PROGRAM P11_E3508
VAR_INPUT
	nTemperatureTargetValue	: INT(0..1200); //Target Values, Input Range 0 ~ 1200 Celcius
	nRampTime				: INT := 1; //Second
	nPowerRateSetValue		: WORD;	
	bOutputManAuto 			: BOOL; // 0:Auto, 1:Manual Operation
	
	bHeaterOn				: BOOL := FALSE; //to PSTEK
	bHeaterReset			: BOOL; //to PSTEK

END_VAR
VAR_OUTPUT
	bAlarmState_E3508 		: BOOL; //Alarm or Sensor Break Signal
	bManAuto_E3508 			: BOOL; // 0:Manual, 1:Auto
	rPowerRate				: REAL;	//Power rate for Monitoring
	
	isHeaterReady			: BOOL; //Close : Ready
	isHeaterRun				: BOOL; //Close : Running, Open : Stop
	isHeaterFault			: BOOL; //Close : Falut, Open : Normal
	//isInductionHeaterErr	: BOOL; //Power Supply
	bInductionHeaterCB		: BOOL;
END_VAR

VAR
	//Input from E3508 Controller
	aInputPVBytes AT %I* 		: ARRAY[1..2]OF USINT; //Input Process Values
	aInputSVBytes AT %I* 		: ARRAY[1..2]OF USINT; //Input Set Values
	aInputTVBytes AT %I* 		: ARRAY[1..2]OF USINT; //Input Target Valuse
	aInputCVBytes AT %I* 		: ARRAY[1..2]OF USINT; //Induction Heter Controlled Values
	aInputProportional AT %I* 	: ARRAY[1..2]OF USINT; //PID - Proportional Band
	aInputIntegral AT %I* 		: ARRAY[1..2]OF USINT; //PID - Integral Time
	aInputDerivative AT %I* 	: ARRAY[1..2]OF USINT; //PID - Derivative Time 
	nInputAlarmBytes AT %I* 	: USINT; // Alarm State
	nInputManAutoBytes AT %I* 	: USINT; // ManAuto State
	
	nTemperaturePV_E3508		: WORD;
	nTemperatureSV_E3508		: WORD;
	nPowerRate_E3508		: WORD; //To Induction Heater Control Values
	nParameterP				: WORD; //PID Parameter P
	nParameterI				: WORD; //PID Parameter I
	nParameterD				: WORD; //PID Parameter D
	//Output to E3508 Controller
	wOutputSVBytes 				: outWord;
	wOutputPowerSVBytes 		: outWord;
	aOutputSVBytes AT %Q* 		: ARRAY[1..2]OF USINT; //Temperature Set Value
	nOutputManAutoBytes AT %Q* 	: USINT; //ManAuto Change
	aOutputPowerBytes AT %Q* 	: ARRAY[1..2]OF USINT; //Output Power in Manual State
	//nOutputAlarmClear AT %Q* : USINT; //Alarm Clear Set
	
	nTemperatureControlValue	: WORD;
	
	// for FB_CTRL_RAMP_GENERATOR Variable
	(* input *)
	bEnable					: BOOL;
	rTemperatureStartValue	: REAL;
	rTemperatureTargetValue	: REAL;
	(* output *)
	rTemperatureControlValue : LREAL;
	bValueReached			: BOOL;
	(* function block *)
	fbCTRL_RAMP_GENERATOR		: FB_CTRL_RAMP_GENERATOR;
	stCTRL_RAMP_GENERATOR_PARAMS: ST_CTRL_RAMP_GENERATOR_PARAMS;

	eErrorId				: E_CTRL_ERRORCODES;
	bError					: BOOL;
	bInit					: BOOL := TRUE;

	(* Induction Heating Operation Parameter*)
	rRampingRatio			: REAL;	
END_VAR

//Induction Heater & Temperature Controller & Thermo Couple(R-Type)
//Maker: PSTEK, Eurotherm
//Model: 3508
//Temperature Range: 0 ~ 12000℃

(* Read from Power Distribution Pannel *)
bInductionHeaterCB		:= GVL_IO.aDigitalInputIO[4].7;

(* Read from E3508 Device Value *)
nTemperaturePV_E3508	:= USINT_TO_WORD_Bit(aInputPVBytes[1], aInputPVBytes[2]);
nTemperatureSV_E3508	:= USINT_TO_WORD_Bit(aInputSVBytes[1], aInputSVBytes[2]);
nPowerRate_E3508		:= USINT_TO_WORD_Bit(aInputCVBytes[1], aInputCVBytes[2]); //divided to 10
nParameterP 			:= USINT_TO_WORD_Bit(aInputProportional[1], aInputProportional[2]);
nParameterI 			:= USINT_TO_WORD_Bit(aInputIntegral[1], aInputIntegral[2]);
nParameterD 			:= USINT_TO_WORD_Bit(aInputDerivative[1], aInputDerivative[2]);

bAlarmState_E3508 		:= nInputAlarmBytes.7;
bManAuto_E3508 			:= nInputManAutoBytes.7;

(* Read from Induction Heater Value *)
isHeaterReady 			:= GVL_IO.aDigitalInputIO[2].2;
isHeaterRun		 		:= GVL_IO.aDigitalInputIO[2].3;
isHeaterFault 			:= GVL_IO.aDigitalInputIO[2].4;

(*Ramp Generator Parameter Variable*)
rTemperatureTargetValue	:= INT_TO_REAL(nTemperatureTargetValue);
rPowerRate				:= WORD_TO_REAL(nPowerRate_E3508)*0.1; //divided to 10

bHeaterOn := TRUE;
bInit := NOT((rTemperatureTargetValue = 0) AND (rTemperatureStartValue = 0));

IF bInit AND nRampTime <> 0 AND RCP.iRcpOperationState=10 THEN
	rRampingRatio := ABS(rTemperatureTargetValue - rTemperatureStartValue) / nRampTime; //Second
	(* init parameter struct *)
	stCTRL_RAMP_GENERATOR_PARAMS.tTaskCycleTime		:= T#2MS;
	stCTRL_RAMP_GENERATOR_PARAMS.tCtrlCycleTime		:= T#100MS;
	stCTRL_RAMP_GENERATOR_PARAMS.fVeloPos			:= rRampingRatio; (* in units per second *)
	stCTRL_RAMP_GENERATOR_PARAMS.fVeloNeg			:= rRampingRatio; (* in units per second *)

	IF rTemperatureTargetValue <> rTemperatureStartValue THEN
		bEnable := TRUE;
		(* call function block *)
		fbCTRL_RAMP_GENERATOR(
			bEnable			:= bEnable,
			fStart			:= rTemperatureStartValue,
			fTarget			:= rTemperatureTargetValue,
			stParams		:= stCTRL_RAMP_GENERATOR_PARAMS,
			fOut			=> rTemperatureControlValue,
			bValueReached	=> bValueReached,
			bError			=> bError,
			eErrorId		=> eErrorId);
	ELSE
		fbCTRL_RAMP_GENERATOR.bEnable := FALSE;
	END_IF

	IF bValueReached THEN
		rTemperatureStartValue	:= LREAL_TO_REAL(rTemperatureControlValue);
	END_IF
END_IF

nTemperatureControlValue	:= LREAL_TO_WORD(rTemperatureControlValue);

(* Write to E3508 Device Value *)
wOutputSVBytes 			:= WORD_TO_USINT_Bit(nTemperatureControlValue);
aOutputSVBytes[1] 		:= wOutputSVBytes.Lower;
aOutputSVBytes[2] 		:= wOutputSVBytes.Upper;

// PowerRate Operation
nOutputManAutoBytes.0 	:= bOutputManAuto;

wOutputPowerSVBytes 	:= WORD_TO_USINT_Bit(nPowerRateSetValue*10); //multiple to 10
aOutputPowerBytes[1] 	:= wOutputPowerSVBytes.Lower;
aOutputPowerBytes[2] 	:= wOutputPowerSVBytes.Upper;

(* Write to Induction Heater Value *)
GVL_IO.aDigitalOutputIO[2].0 := bHeaterOn;
GVL_IO.aDigitalOutputIO[2].1 := bHeaterReset;

END_PROGRAM

(* stored: Version 1.1.0.1, ProductVersion 3.1.4026.8
   POU P11_E3508: Id {a7e3d6a1-82f0-4607-8ac9-093cb5f931f5}, SpecialFunc None *)
